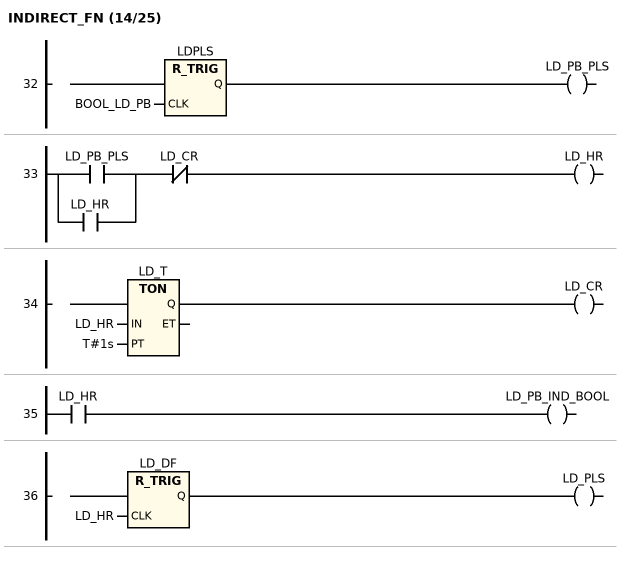
// NETWORK 32
LDPLS(CLK := BOOL_LD_PB); // R_TRIG
LD_PB_PLS := LDPLS.Q;

// NETWORK 33
LD_HR := (LD_PB_PLS OR LD_HR) AND NOT LD_CR;

// NETWORK 34
LD_T(IN := LD_HR, PT := T#1s); // TON
LD_CR := LD_T.Q;

// NETWORK 35
LD_PB_IND_BOOL := LD_HR;

// NETWORK 36
LD_DF(CLK := LD_HR); // R_TRIG
LD_PLS := LD_DF.Q;

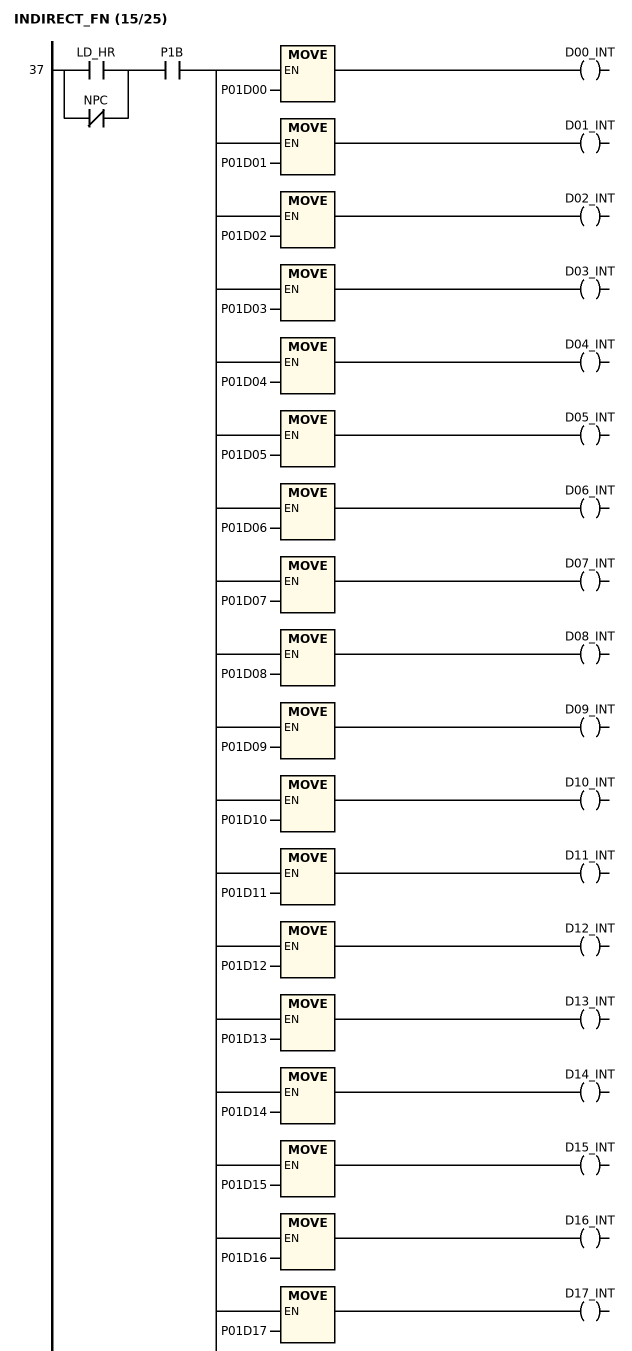
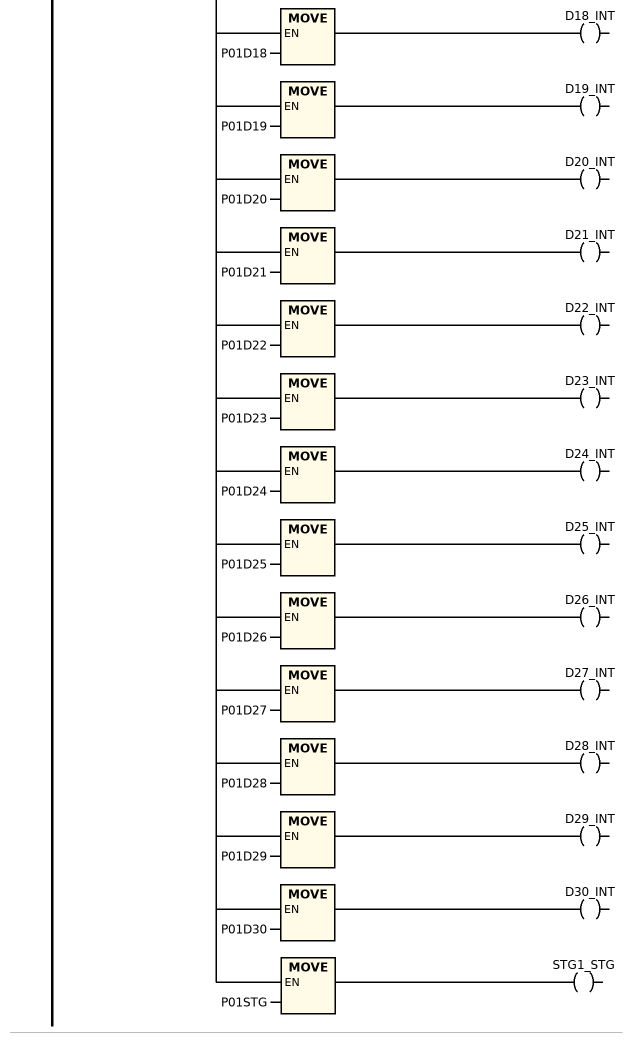
// NETWORK 37
_w365 := (LD_HR OR NOT NPC) AND P1B;
IF _w365 THEN _w366 := P01D00; END_IF
D00_INT := _w366;
IF _w365 THEN _w367 := P01D01; END_IF
D01_INT := _w367;
IF _w365 THEN _w368 := P01D02; END_IF
D02_INT := _w368;
IF _w365 THEN _w369 := P01D03; END_IF
D03_INT := _w369;
IF _w365 THEN _w370 := P01D04; END_IF
D04_INT := _w370;
IF _w365 THEN _w371 := P01D05; END_IF
D05_INT := _w371;
IF _w365 THEN _w372 := P01D06; END_IF
D06_INT := _w372;
IF _w365 THEN _w373 := P01D07; END_IF
D07_INT := _w373;
IF _w365 THEN _w374 := P01D08; END_IF
D08_INT := _w374;
IF _w365 THEN _w375 := P01D09; END_IF
D09_INT := _w375;
IF _w365 THEN _w376 := P01D10; END_IF
D10_INT := _w376;
IF _w365 THEN _w377 := P01D11; END_IF
D11_INT := _w377;
IF _w365 THEN _w378 := P01D12; END_IF
D12_INT := _w378;
IF _w365 THEN _w379 := P01D13; END_IF
D13_INT := _w379;
IF _w365 THEN _w380 := P01D14; END_IF
D14_INT := _w380;
IF _w365 THEN _w381 := P01D15; END_IF
D15_INT := _w381;
IF _w365 THEN _w382 := P01D16; END_IF
D16_INT := _w382;
IF _w365 THEN _w383 := P01D17; END_IF
D17_INT := _w383;
IF _w365 THEN _w384 := P01D18; END_IF
D18_INT := _w384;
IF _w365 THEN _w385 := P01D19; END_IF
D19_INT := _w385;
IF _w365 THEN _w386 := P01D20; END_IF
D20_INT := _w386;
IF _w365 THEN _w387 := P01D21; END_IF
D21_INT := _w387;
IF _w365 THEN _w388 := P01D22; END_IF
D22_INT := _w388;
IF _w365 THEN _w389 := P01D23; END_IF
D23_INT := _w389;
IF _w365 THEN _w390 := P01D24; END_IF
D24_INT := _w390;
IF _w365 THEN _w391 := P01D25; END_IF
D25_INT := _w391;
IF _w365 THEN _w392 := P01D26; END_IF
D26_INT := _w392;
IF _w365 THEN _w393 := P01D27; END_IF
D27_INT := _w393;
IF _w365 THEN _w394 := P01D28; END_IF
D28_INT := _w394;
IF _w365 THEN _w395 := P01D29; END_IF
D29_INT := _w395;
IF _w365 THEN _w396 := P01D30; END_IF
D30_INT := _w396;
IF _w365 THEN _w397 := P01STG; END_IF
STG1_STG := _w397;

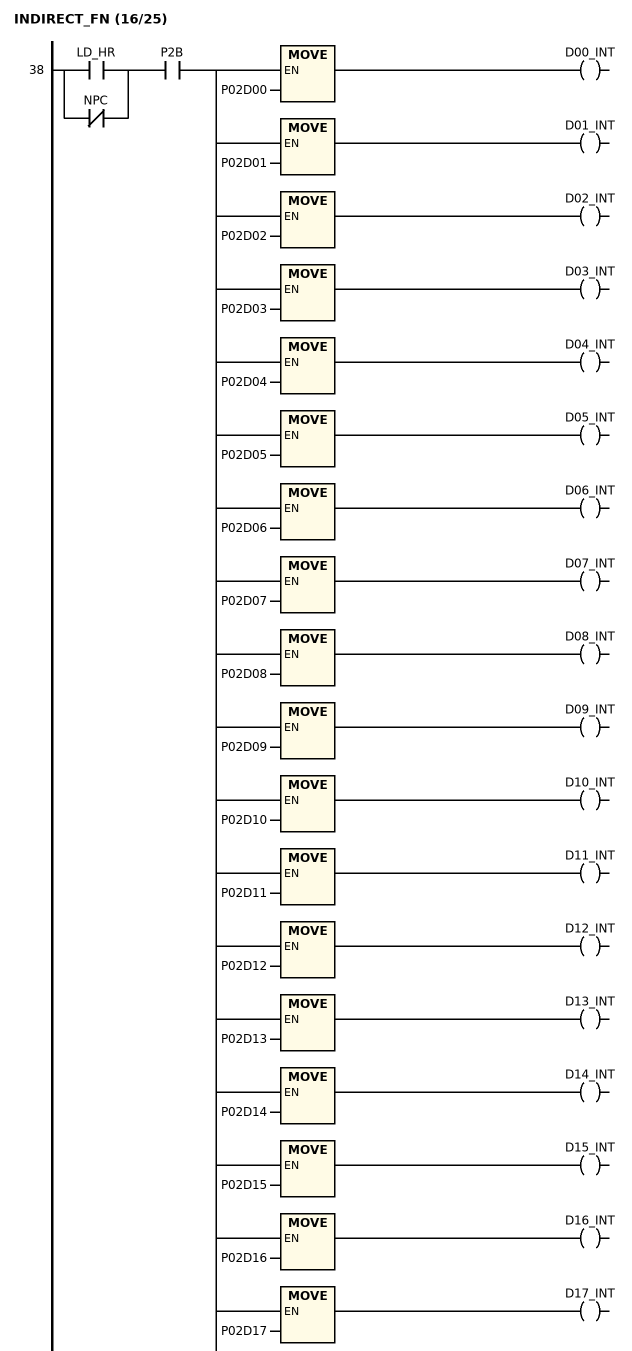
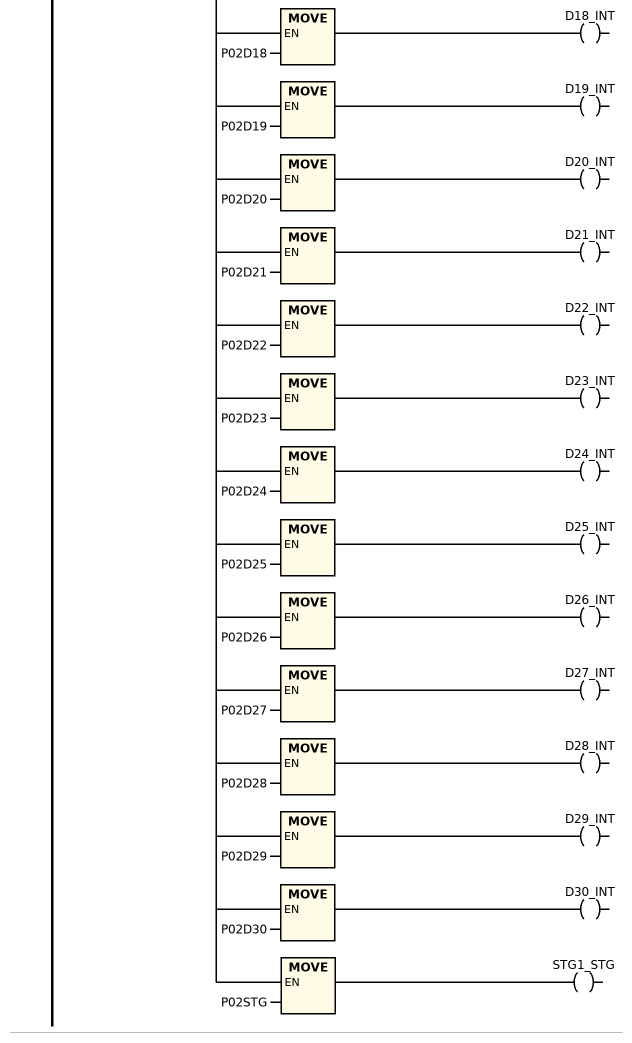
// NETWORK 38
_w398 := (LD_HR OR NOT NPC) AND P2B;
IF _w398 THEN _w399 := P02D00; END_IF
D00_INT := _w399;
IF _w398 THEN _w400 := P02D01; END_IF
D01_INT := _w400;
IF _w398 THEN _w401 := P02D02; END_IF
D02_INT := _w401;
IF _w398 THEN _w402 := P02D03; END_IF
D03_INT := _w402;
IF _w398 THEN _w403 := P02D04; END_IF
D04_INT := _w403;
IF _w398 THEN _w404 := P02D05; END_IF
D05_INT := _w404;
IF _w398 THEN _w405 := P02D06; END_IF
D06_INT := _w405;
IF _w398 THEN _w406 := P02D07; END_IF
D07_INT := _w406;
IF _w398 THEN _w407 := P02D08; END_IF
D08_INT := _w407;
IF _w398 THEN _w408 := P02D09; END_IF
D09_INT := _w408;
IF _w398 THEN _w409 := P02D10; END_IF
D10_INT := _w409;
IF _w398 THEN _w410 := P02D11; END_IF
D11_INT := _w410;
IF _w398 THEN _w411 := P02D12; END_IF
D12_INT := _w411;
IF _w398 THEN _w412 := P02D13; END_IF
D13_INT := _w412;
IF _w398 THEN _w413 := P02D14; END_IF
D14_INT := _w413;
IF _w398 THEN _w414 := P02D15; END_IF
D15_INT := _w414;
IF _w398 THEN _w415 := P02D16; END_IF
D16_INT := _w415;
IF _w398 THEN _w416 := P02D17; END_IF
D17_INT := _w416;
IF _w398 THEN _w417 := P02D18; END_IF
D18_INT := _w417;
IF _w398 THEN _w418 := P02D19; END_IF
D19_INT := _w418;
IF _w398 THEN _w419 := P02D20; END_IF
D20_INT := _w419;
IF _w398 THEN _w420 := P02D21; END_IF
D21_INT := _w420;
IF _w398 THEN _w421 := P02D22; END_IF
D22_INT := _w421;
IF _w398 THEN _w422 := P02D23; END_IF
D23_INT := _w422;
IF _w398 THEN _w423 := P02D24; END_IF
D24_INT := _w423;
IF _w398 THEN _w424 := P02D25; END_IF
D25_INT := _w424;
IF _w398 THEN _w425 := P02D26; END_IF
D26_INT := _w425;
IF _w398 THEN _w426 := P02D27; END_IF
D27_INT := _w426;
IF _w398 THEN _w427 := P02D28; END_IF
D28_INT := _w427;
IF _w398 THEN _w428 := P02D29; END_IF
D29_INT := _w428;
IF _w398 THEN _w429 := P02D30; END_IF
D30_INT := _w429;
IF _w398 THEN _w430 := P02STG; END_IF
STG1_STG := _w430;

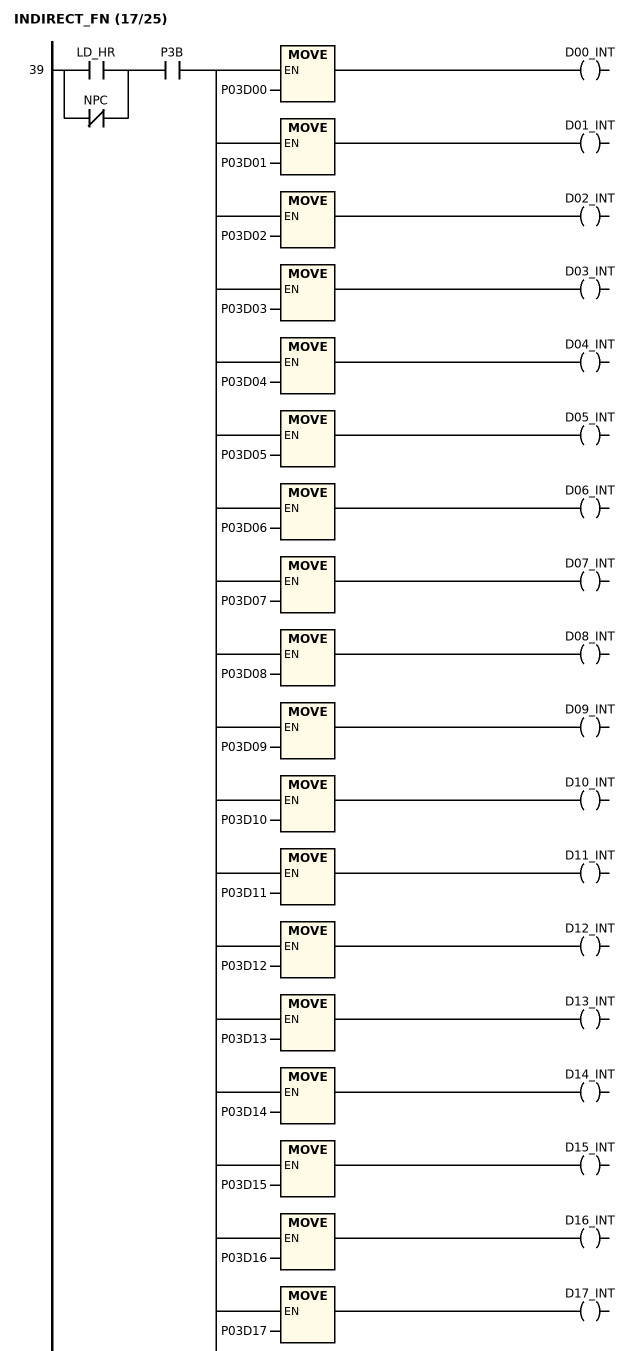
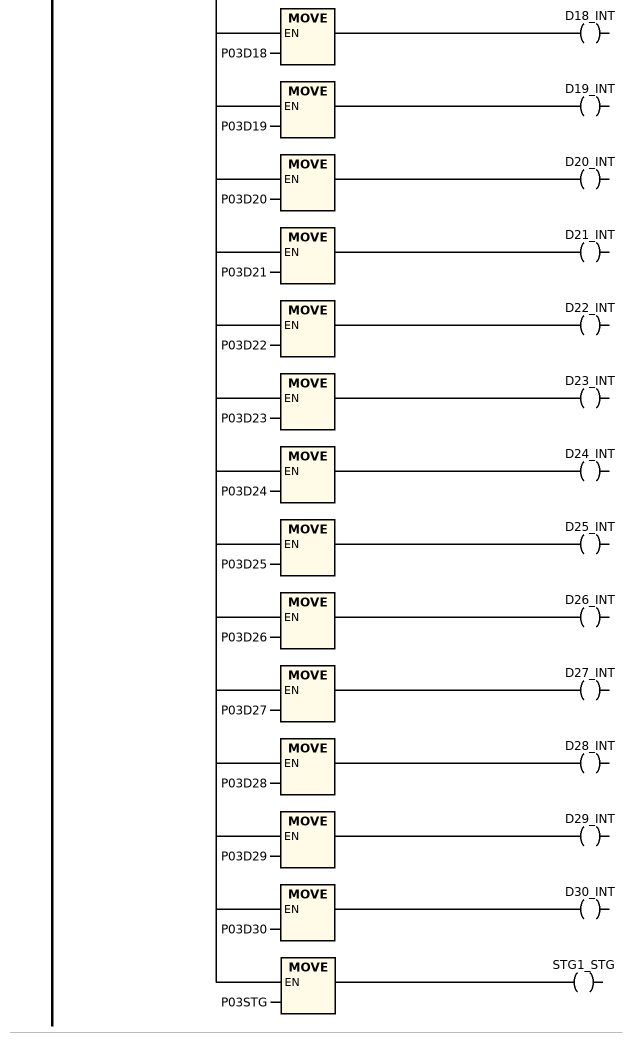
// NETWORK 39
_w431 := (LD_HR OR NOT NPC) AND P3B;
IF _w431 THEN _w432 := P03D00; END_IF
D00_INT := _w432;
IF _w431 THEN _w433 := P03D01; END_IF
D01_INT := _w433;
IF _w431 THEN _w434 := P03D02; END_IF
D02_INT := _w434;
IF _w431 THEN _w435 := P03D03; END_IF
D03_INT := _w435;
IF _w431 THEN _w436 := P03D04; END_IF
D04_INT := _w436;
IF _w431 THEN _w437 := P03D05; END_IF
D05_INT := _w437;
IF _w431 THEN _w438 := P03D06; END_IF
D06_INT := _w438;
IF _w431 THEN _w439 := P03D07; END_IF
D07_INT := _w439;
IF _w431 THEN _w440 := P03D08; END_IF
D08_INT := _w440;
IF _w431 THEN _w441 := P03D09; END_IF
D09_INT := _w441;
IF _w431 THEN _w442 := P03D10; END_IF
D10_INT := _w442;
IF _w431 THEN _w443 := P03D11; END_IF
D11_INT := _w443;
IF _w431 THEN _w444 := P03D12; END_IF
D12_INT := _w444;
IF _w431 THEN _w445 := P03D13; END_IF
D13_INT := _w445;
IF _w431 THEN _w446 := P03D14; END_IF
D14_INT := _w446;
IF _w431 THEN _w447 := P03D15; END_IF
D15_INT := _w447;
IF _w431 THEN _w448 := P03D16; END_IF
D16_INT := _w448;
IF _w431 THEN _w449 := P03D17; END_IF
D17_INT := _w449;
IF _w431 THEN _w450 := P03D18; END_IF
D18_INT := _w450;
IF _w431 THEN _w451 := P03D19; END_IF
D19_INT := _w451;
IF _w431 THEN _w452 := P03D20; END_IF
D20_INT := _w452;
IF _w431 THEN _w453 := P03D21; END_IF
D21_INT := _w453;
IF _w431 THEN _w454 := P03D22; END_IF
D22_INT := _w454;
IF _w431 THEN _w455 := P03D23; END_IF
D23_INT := _w455;
IF _w431 THEN _w456 := P03D24; END_IF
D24_INT := _w456;
IF _w431 THEN _w457 := P03D25; END_IF
D25_INT := _w457;
IF _w431 THEN _w458 := P03D26; END_IF
D26_INT := _w458;
IF _w431 THEN _w459 := P03D27; END_IF
D27_INT := _w459;
IF _w431 THEN _w460 := P03D28; END_IF
D28_INT := _w460;
IF _w431 THEN _w461 := P03D29; END_IF
D29_INT := _w461;
IF _w431 THEN _w462 := P03D30; END_IF
D30_INT := _w462;
IF _w431 THEN _w463 := P03STG; END_IF
STG1_STG := _w463;

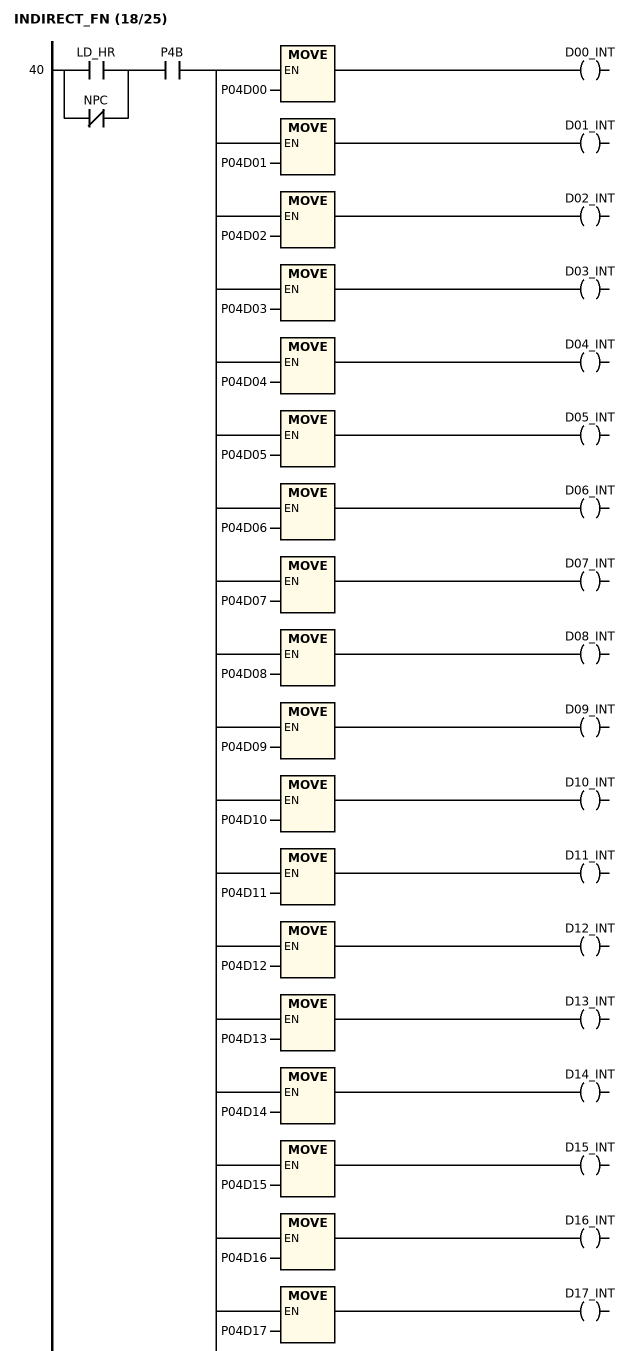
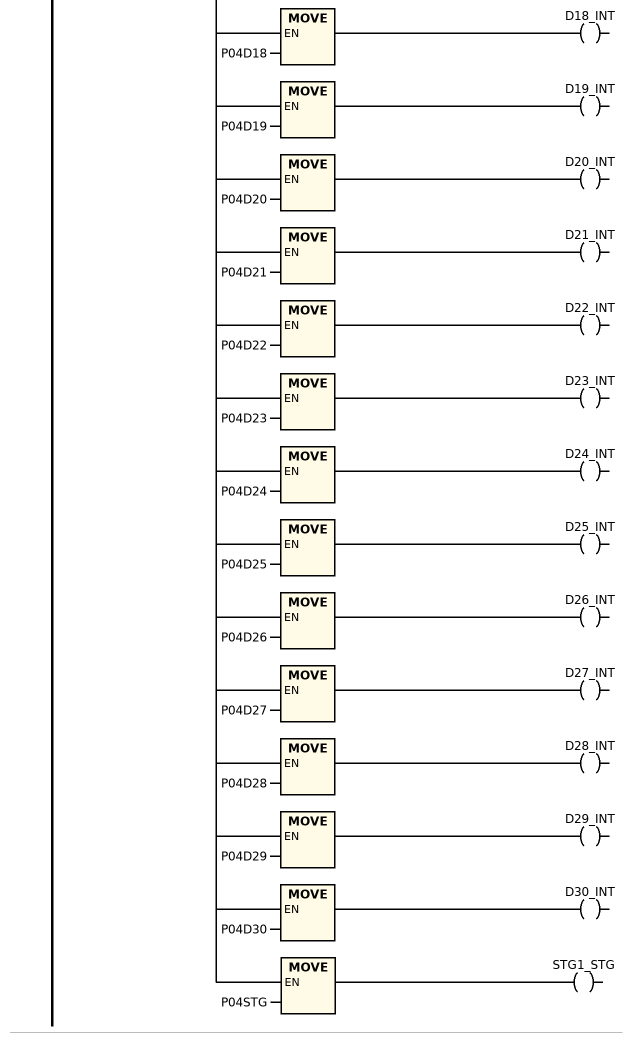
// NETWORK 40
_w464 := (LD_HR OR NOT NPC) AND P4B;
IF _w464 THEN _w465 := P04D00; END_IF
D00_INT := _w465;
IF _w464 THEN _w466 := P04D01; END_IF
D01_INT := _w466;
IF _w464 THEN _w467 := P04D02; END_IF
D02_INT := _w467;
IF _w464 THEN _w468 := P04D03; END_IF
D03_INT := _w468;
IF _w464 THEN _w469 := P04D04; END_IF
D04_INT := _w469;
IF _w464 THEN _w470 := P04D05; END_IF
D05_INT := _w470;
IF _w464 THEN _w471 := P04D06; END_IF
D06_INT := _w471;
IF _w464 THEN _w472 := P04D07; END_IF
D07_INT := _w472;
IF _w464 THEN _w473 := P04D08; END_IF
D08_INT := _w473;
IF _w464 THEN _w474 := P04D09; END_IF
D09_INT := _w474;
IF _w464 THEN _w475 := P04D10; END_IF
D10_INT := _w475;
IF _w464 THEN _w476 := P04D11; END_IF
D11_INT := _w476;
IF _w464 THEN _w477 := P04D12; END_IF
D12_INT := _w477;
IF _w464 THEN _w478 := P04D13; END_IF
D13_INT := _w478;
IF _w464 THEN _w479 := P04D14; END_IF
D14_INT := _w479;
IF _w464 THEN _w480 := P04D15; END_IF
D15_INT := _w480;
IF _w464 THEN _w481 := P04D16; END_IF
D16_INT := _w481;
IF _w464 THEN _w482 := P04D17; END_IF
D17_INT := _w482;
IF _w464 THEN _w483 := P04D18; END_IF
D18_INT := _w483;
IF _w464 THEN _w484 := P04D19; END_IF
D19_INT := _w484;
IF _w464 THEN _w485 := P04D20; END_IF
D20_INT := _w485;
IF _w464 THEN _w486 := P04D21; END_IF
D21_INT := _w486;
IF _w464 THEN _w487 := P04D22; END_IF
D22_INT := _w487;
IF _w464 THEN _w488 := P04D23; END_IF
D23_INT := _w488;
IF _w464 THEN _w489 := P04D24; END_IF
D24_INT := _w489;
IF _w464 THEN _w490 := P04D25; END_IF
D25_INT := _w490;
IF _w464 THEN _w491 := P04D26; END_IF
D26_INT := _w491;
IF _w464 THEN _w492 := P04D27; END_IF
D27_INT := _w492;
IF _w464 THEN _w493 := P04D28; END_IF
D28_INT := _w493;
IF _w464 THEN _w494 := P04D29; END_IF
D29_INT := _w494;
IF _w464 THEN _w495 := P04D30; END_IF
D30_INT := _w495;
IF _w464 THEN _w496 := P04STG; END_IF
STG1_STG := _w496;

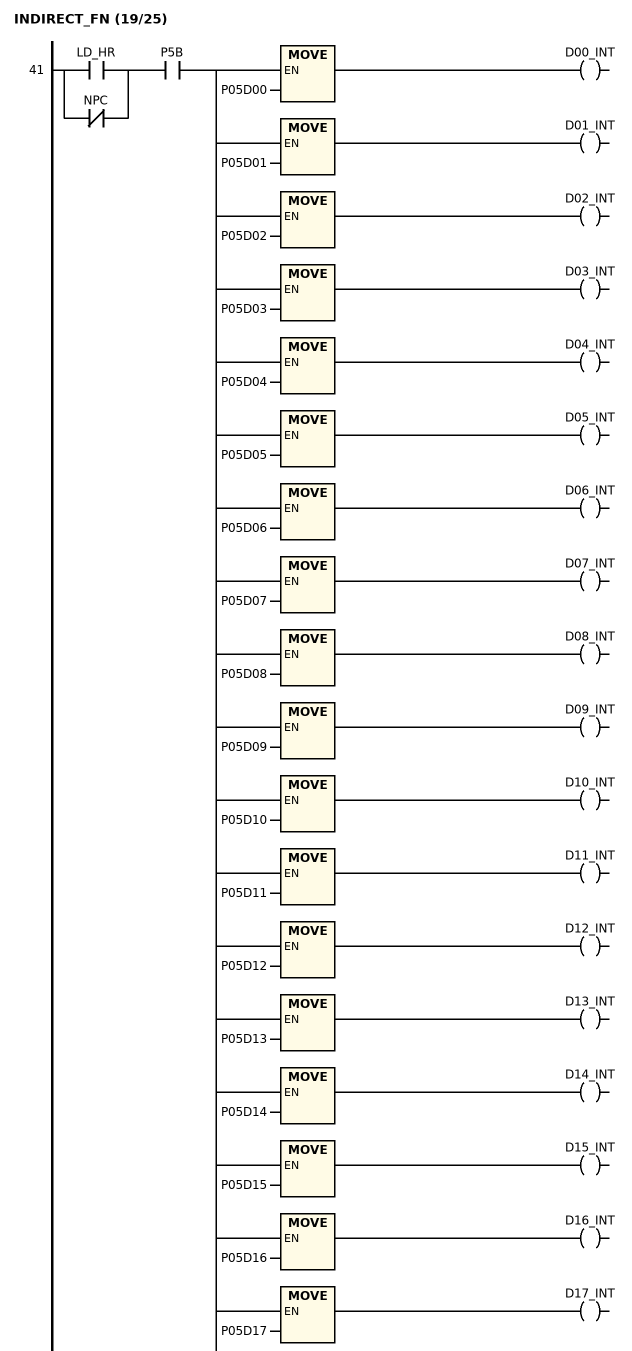
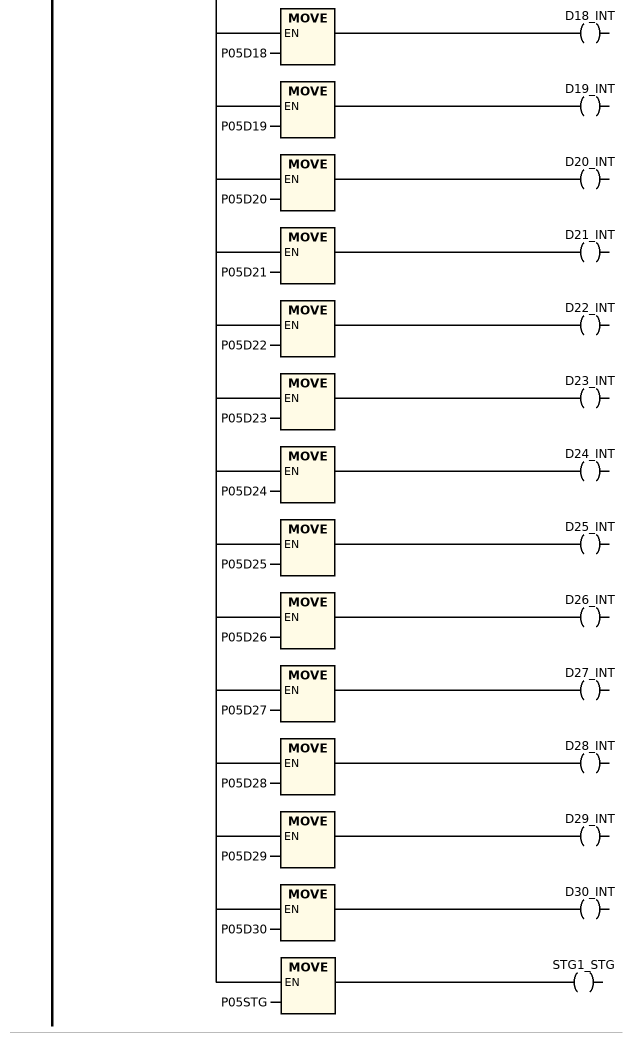
// NETWORK 41
_w497 := (LD_HR OR NOT NPC) AND P5B;
IF _w497 THEN _w498 := P05D00; END_IF
D00_INT := _w498;
IF _w497 THEN _w499 := P05D01; END_IF
D01_INT := _w499;
IF _w497 THEN _w500 := P05D02; END_IF
D02_INT := _w500;
IF _w497 THEN _w501 := P05D03; END_IF
D03_INT := _w501;
IF _w497 THEN _w502 := P05D04; END_IF
D04_INT := _w502;
IF _w497 THEN _w503 := P05D05; END_IF
D05_INT := _w503;
IF _w497 THEN _w504 := P05D06; END_IF
D06_INT := _w504;
IF _w497 THEN _w505 := P05D07; END_IF
D07_INT := _w505;
IF _w497 THEN _w506 := P05D08; END_IF
D08_INT := _w506;
IF _w497 THEN _w507 := P05D09; END_IF
D09_INT := _w507;
IF _w497 THEN _w508 := P05D10; END_IF
D10_INT := _w508;
IF _w497 THEN _w509 := P05D11; END_IF
D11_INT := _w509;
IF _w497 THEN _w510 := P05D12; END_IF
D12_INT := _w510;
IF _w497 THEN _w511 := P05D13; END_IF
D13_INT := _w511;
IF _w497 THEN _w512 := P05D14; END_IF
D14_INT := _w512;
IF _w497 THEN _w513 := P05D15; END_IF
D15_INT := _w513;
IF _w497 THEN _w514 := P05D16; END_IF
D16_INT := _w514;
IF _w497 THEN _w515 := P05D17; END_IF
D17_INT := _w515;
IF _w497 THEN _w516 := P05D18; END_IF
D18_INT := _w516;
IF _w497 THEN _w517 := P05D19; END_IF
D19_INT := _w517;
IF _w497 THEN _w518 := P05D20; END_IF
D20_INT := _w518;
IF _w497 THEN _w519 := P05D21; END_IF
D21_INT := _w519;
IF _w497 THEN _w520 := P05D22; END_IF
D22_INT := _w520;
IF _w497 THEN _w521 := P05D23; END_IF
D23_INT := _w521;
IF _w497 THEN _w522 := P05D24; END_IF
D24_INT := _w522;
IF _w497 THEN _w523 := P05D25; END_IF
D25_INT := _w523;
IF _w497 THEN _w524 := P05D26; END_IF
D26_INT := _w524;
IF _w497 THEN _w525 := P05D27; END_IF
D27_INT := _w525;
IF _w497 THEN _w526 := P05D28; END_IF
D28_INT := _w526;
IF _w497 THEN _w527 := P05D29; END_IF
D29_INT := _w527;
IF _w497 THEN _w528 := P05D30; END_IF
D30_INT := _w528;
IF _w497 THEN _w529 := P05STG; END_IF
STG1_STG := _w529;

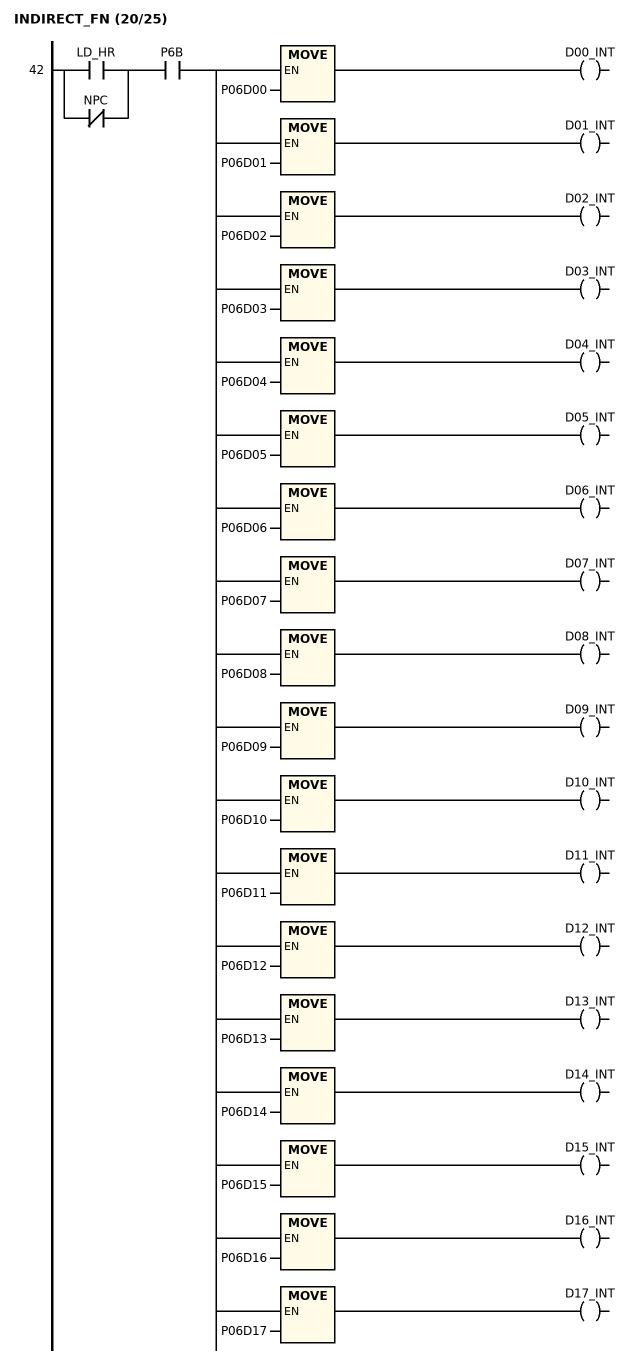
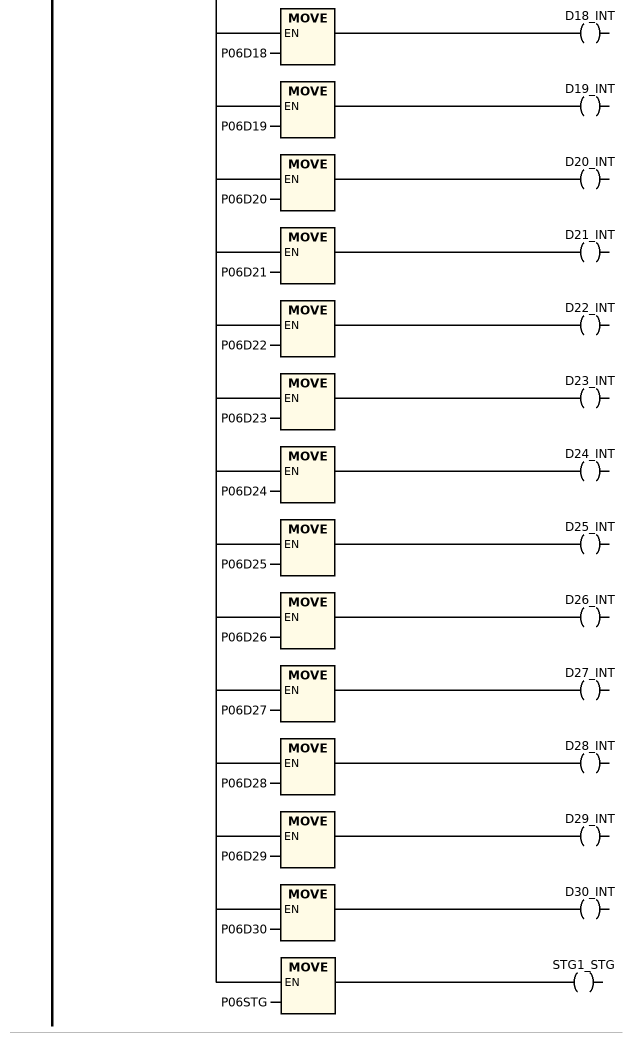
// NETWORK 42
_w530 := (LD_HR OR NOT NPC) AND P6B;
IF _w530 THEN _w531 := P06D00; END_IF
D00_INT := _w531;
IF _w530 THEN _w532 := P06D01; END_IF
D01_INT := _w532;
IF _w530 THEN _w533 := P06D02; END_IF
D02_INT := _w533;
IF _w530 THEN _w534 := P06D03; END_IF
D03_INT := _w534;
IF _w530 THEN _w535 := P06D04; END_IF
D04_INT := _w535;
IF _w530 THEN _w536 := P06D05; END_IF
D05_INT := _w536;
IF _w530 THEN _w537 := P06D06; END_IF
D06_INT := _w537;
IF _w530 THEN _w538 := P06D07; END_IF
D07_INT := _w538;
IF _w530 THEN _w539 := P06D08; END_IF
D08_INT := _w539;
IF _w530 THEN _w540 := P06D09; END_IF
D09_INT := _w540;
IF _w530 THEN _w541 := P06D10; END_IF
D10_INT := _w541;
IF _w530 THEN _w542 := P06D11; END_IF
D11_INT := _w542;
IF _w530 THEN _w543 := P06D12; END_IF
D12_INT := _w543;
IF _w530 THEN _w544 := P06D13; END_IF
D13_INT := _w544;
IF _w530 THEN _w545 := P06D14; END_IF
D14_INT := _w545;
IF _w530 THEN _w546 := P06D15; END_IF
D15_INT := _w546;
IF _w530 THEN _w547 := P06D16; END_IF
D16_INT := _w547;
IF _w530 THEN _w548 := P06D17; END_IF
D17_INT := _w548;
IF _w530 THEN _w549 := P06D18; END_IF
D18_INT := _w549;
IF _w530 THEN _w550 := P06D19; END_IF
D19_INT := _w550;
IF _w530 THEN _w551 := P06D20; END_IF
D20_INT := _w551;
IF _w530 THEN _w552 := P06D21; END_IF
D21_INT := _w552;
IF _w530 THEN _w553 := P06D22; END_IF
D22_INT := _w553;
IF _w530 THEN _w554 := P06D23; END_IF
D23_INT := _w554;
IF _w530 THEN _w555 := P06D24; END_IF
D24_INT := _w555;
IF _w530 THEN _w556 := P06D25; END_IF
D25_INT := _w556;
IF _w530 THEN _w557 := P06D26; END_IF
D26_INT := _w557;
IF _w530 THEN _w558 := P06D27; END_IF
D27_INT := _w558;
IF _w530 THEN _w559 := P06D28; END_IF
D28_INT := _w559;
IF _w530 THEN _w560 := P06D29; END_IF
D29_INT := _w560;
IF _w530 THEN _w561 := P06D30; END_IF
D30_INT := _w561;
IF _w530 THEN _w562 := P06STG; END_IF
STG1_STG := _w562;

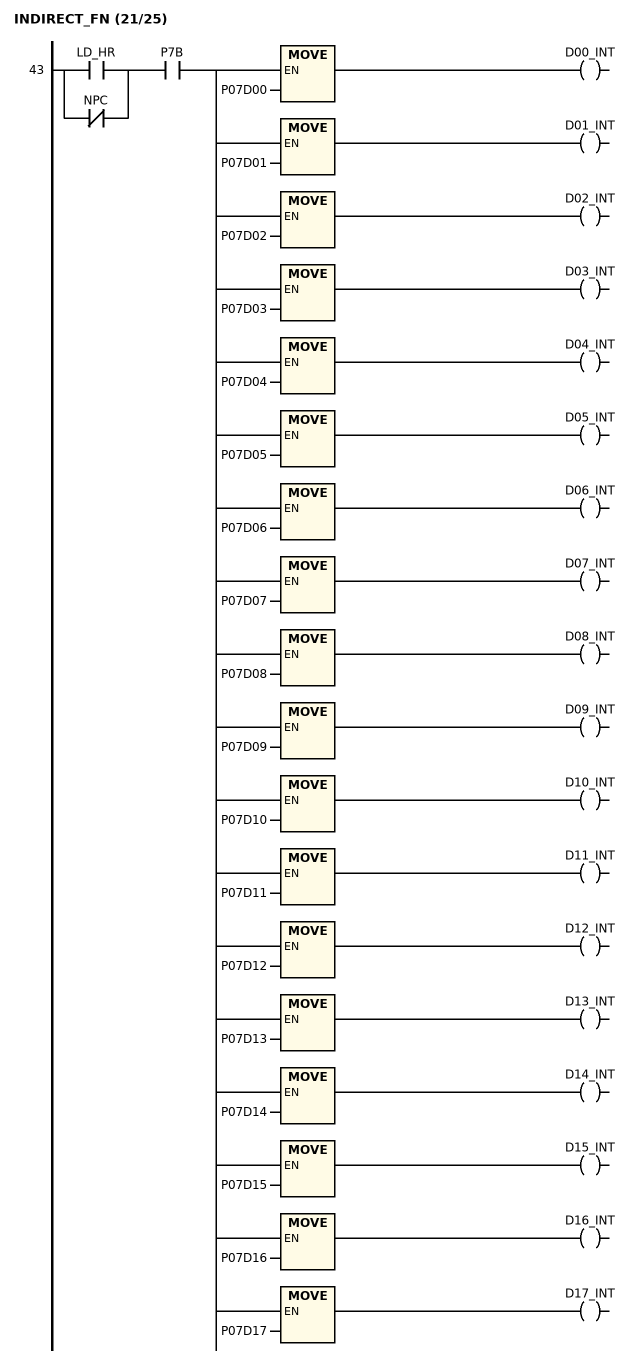
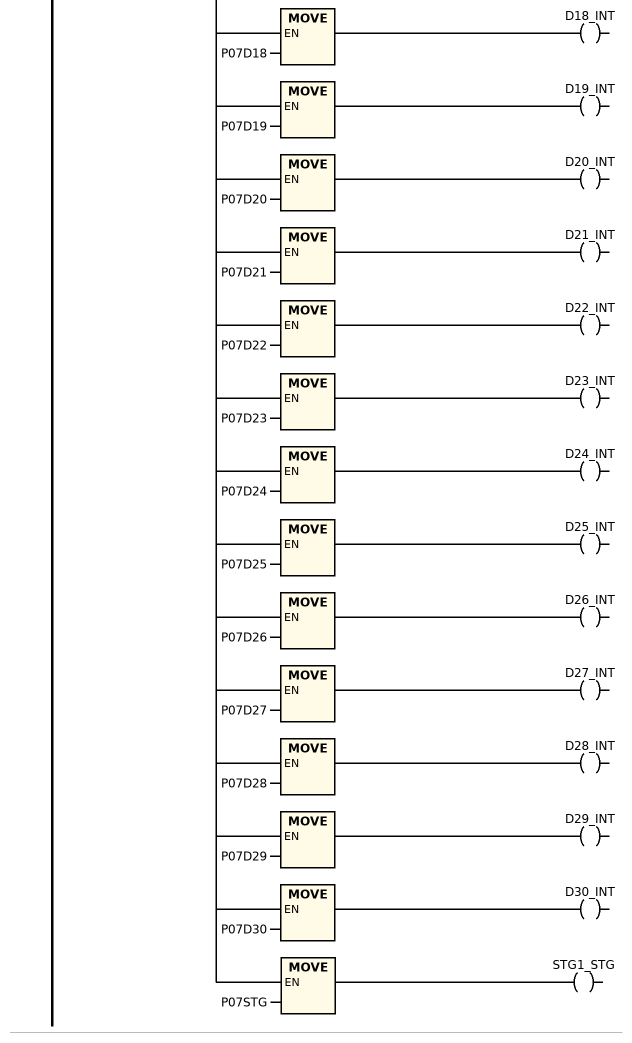
// NETWORK 43
_w563 := (LD_HR OR NOT NPC) AND P7B;
IF _w563 THEN _w564 := P07D00; END_IF
D00_INT := _w564;
IF _w563 THEN _w565 := P07D01; END_IF
D01_INT := _w565;
IF _w563 THEN _w566 := P07D02; END_IF
D02_INT := _w566;
IF _w563 THEN _w567 := P07D03; END_IF
D03_INT := _w567;
IF _w563 THEN _w568 := P07D04; END_IF
D04_INT := _w568;
IF _w563 THEN _w569 := P07D05; END_IF
D05_INT := _w569;
IF _w563 THEN _w570 := P07D06; END_IF
D06_INT := _w570;
IF _w563 THEN _w571 := P07D07; END_IF
D07_INT := _w571;
IF _w563 THEN _w572 := P07D08; END_IF
D08_INT := _w572;
IF _w563 THEN _w573 := P07D09; END_IF
D09_INT := _w573;
IF _w563 THEN _w574 := P07D10; END_IF
D10_INT := _w574;
IF _w563 THEN _w575 := P07D11; END_IF
D11_INT := _w575;
IF _w563 THEN _w576 := P07D12; END_IF
D12_INT := _w576;
IF _w563 THEN _w577 := P07D13; END_IF
D13_INT := _w577;
IF _w563 THEN _w578 := P07D14; END_IF
D14_INT := _w578;
IF _w563 THEN _w579 := P07D15; END_IF
D15_INT := _w579;
IF _w563 THEN _w580 := P07D16; END_IF
D16_INT := _w580;
IF _w563 THEN _w581 := P07D17; END_IF
D17_INT := _w581;
IF _w563 THEN _w582 := P07D18; END_IF
D18_INT := _w582;
IF _w563 THEN _w583 := P07D19; END_IF
D19_INT := _w583;
IF _w563 THEN _w584 := P07D20; END_IF
D20_INT := _w584;
IF _w563 THEN _w585 := P07D21; END_IF
D21_INT := _w585;
IF _w563 THEN _w586 := P07D22; END_IF
D22_INT := _w586;
IF _w563 THEN _w587 := P07D23; END_IF
D23_INT := _w587;
IF _w563 THEN _w588 := P07D24; END_IF
D24_INT := _w588;
IF _w563 THEN _w589 := P07D25; END_IF
D25_INT := _w589;
IF _w563 THEN _w590 := P07D26; END_IF
D26_INT := _w590;
IF _w563 THEN _w591 := P07D27; END_IF
D27_INT := _w591;
IF _w563 THEN _w592 := P07D28; END_IF
D28_INT := _w592;
IF _w563 THEN _w593 := P07D29; END_IF
D29_INT := _w593;
IF _w563 THEN _w594 := P07D30; END_IF
D30_INT := _w594;
IF _w563 THEN _w595 := P07STG; END_IF
STG1_STG := _w595;

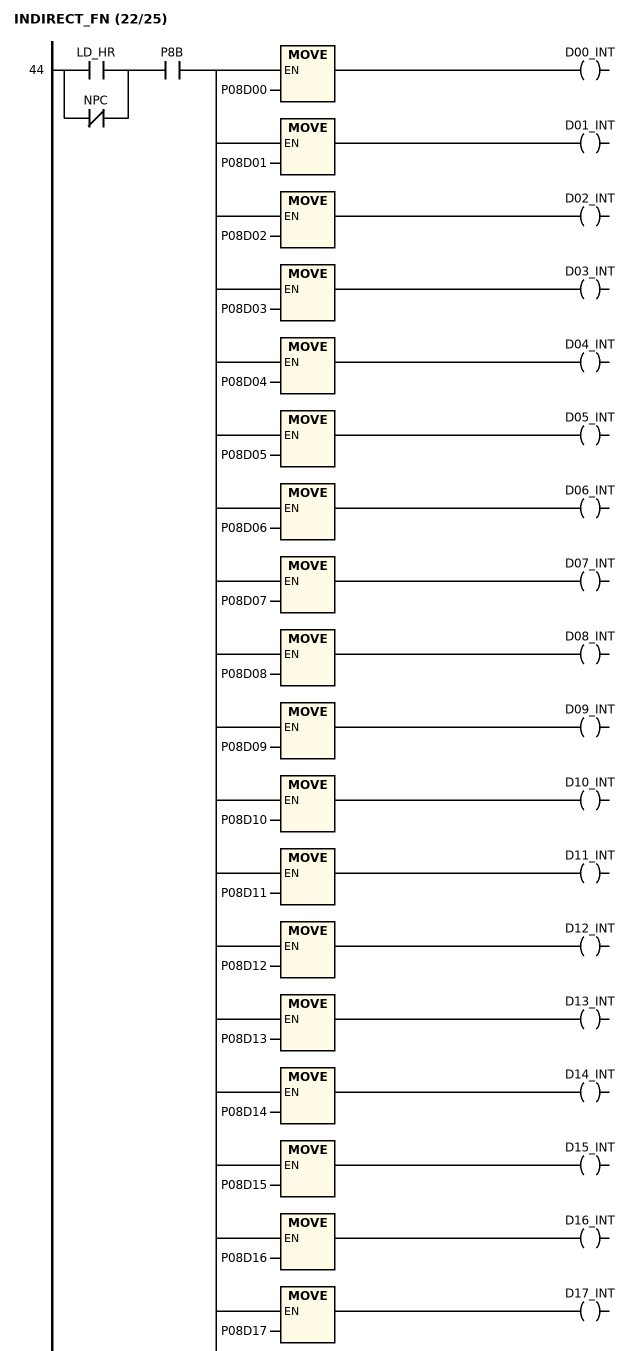
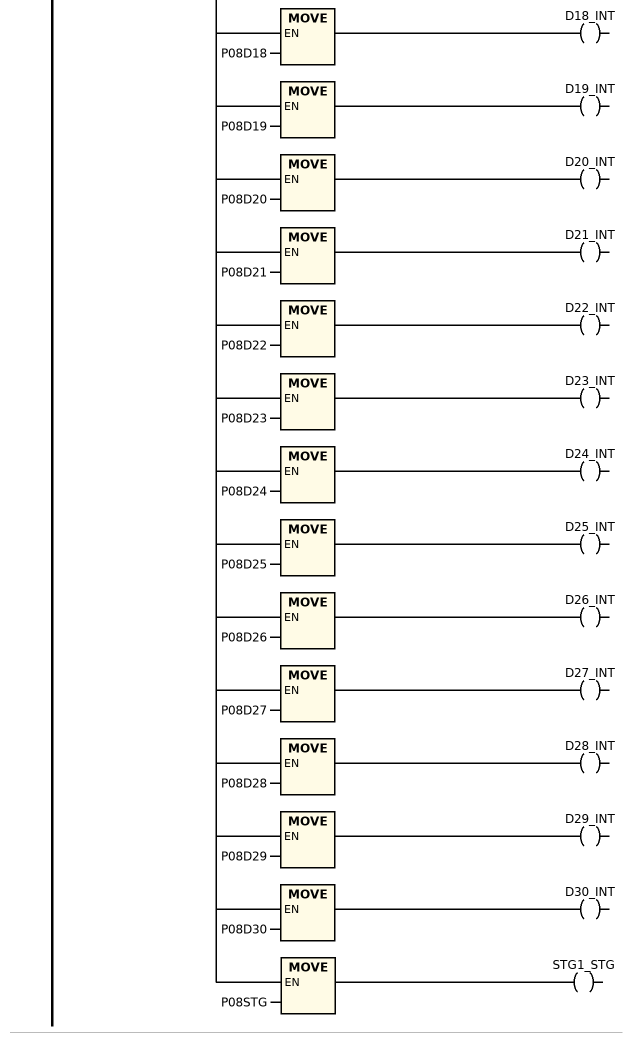
// NETWORK 44
_w596 := (LD_HR OR NOT NPC) AND P8B;
IF _w596 THEN _w597 := P08D00; END_IF
D00_INT := _w597;
IF _w596 THEN _w598 := P08D01; END_IF
D01_INT := _w598;
IF _w596 THEN _w599 := P08D02; END_IF
D02_INT := _w599;
IF _w596 THEN _w600 := P08D03; END_IF
D03_INT := _w600;
IF _w596 THEN _w601 := P08D04; END_IF
D04_INT := _w601;
IF _w596 THEN _w602 := P08D05; END_IF
D05_INT := _w602;
IF _w596 THEN _w603 := P08D06; END_IF
D06_INT := _w603;
IF _w596 THEN _w604 := P08D07; END_IF
D07_INT := _w604;
IF _w596 THEN _w605 := P08D08; END_IF
D08_INT := _w605;
IF _w596 THEN _w606 := P08D09; END_IF
D09_INT := _w606;
IF _w596 THEN _w607 := P08D10; END_IF
D10_INT := _w607;
IF _w596 THEN _w608 := P08D11; END_IF
D11_INT := _w608;
IF _w596 THEN _w609 := P08D12; END_IF
D12_INT := _w609;
IF _w596 THEN _w610 := P08D13; END_IF
D13_INT := _w610;
IF _w596 THEN _w611 := P08D14; END_IF
D14_INT := _w611;
IF _w596 THEN _w612 := P08D15; END_IF
D15_INT := _w612;
IF _w596 THEN _w613 := P08D16; END_IF
D16_INT := _w613;
IF _w596 THEN _w614 := P08D17; END_IF
D17_INT := _w614;
IF _w596 THEN _w615 := P08D18; END_IF
D18_INT := _w615;
IF _w596 THEN _w616 := P08D19; END_IF
D19_INT := _w616;
IF _w596 THEN _w617 := P08D20; END_IF
D20_INT := _w617;
IF _w596 THEN _w618 := P08D21; END_IF
D21_INT := _w618;
IF _w596 THEN _w619 := P08D22; END_IF
D22_INT := _w619;
IF _w596 THEN _w620 := P08D23; END_IF
D23_INT := _w620;
IF _w596 THEN _w621 := P08D24; END_IF
D24_INT := _w621;
IF _w596 THEN _w622 := P08D25; END_IF
D25_INT := _w622;
IF _w596 THEN _w623 := P08D26; END_IF
D26_INT := _w623;
IF _w596 THEN _w624 := P08D27; END_IF
D27_INT := _w624;
IF _w596 THEN _w625 := P08D28; END_IF
D28_INT := _w625;
IF _w596 THEN _w626 := P08D29; END_IF
D29_INT := _w626;
IF _w596 THEN _w627 := P08D30; END_IF
D30_INT := _w627;
IF _w596 THEN _w628 := P08STG; END_IF
STG1_STG := _w628;

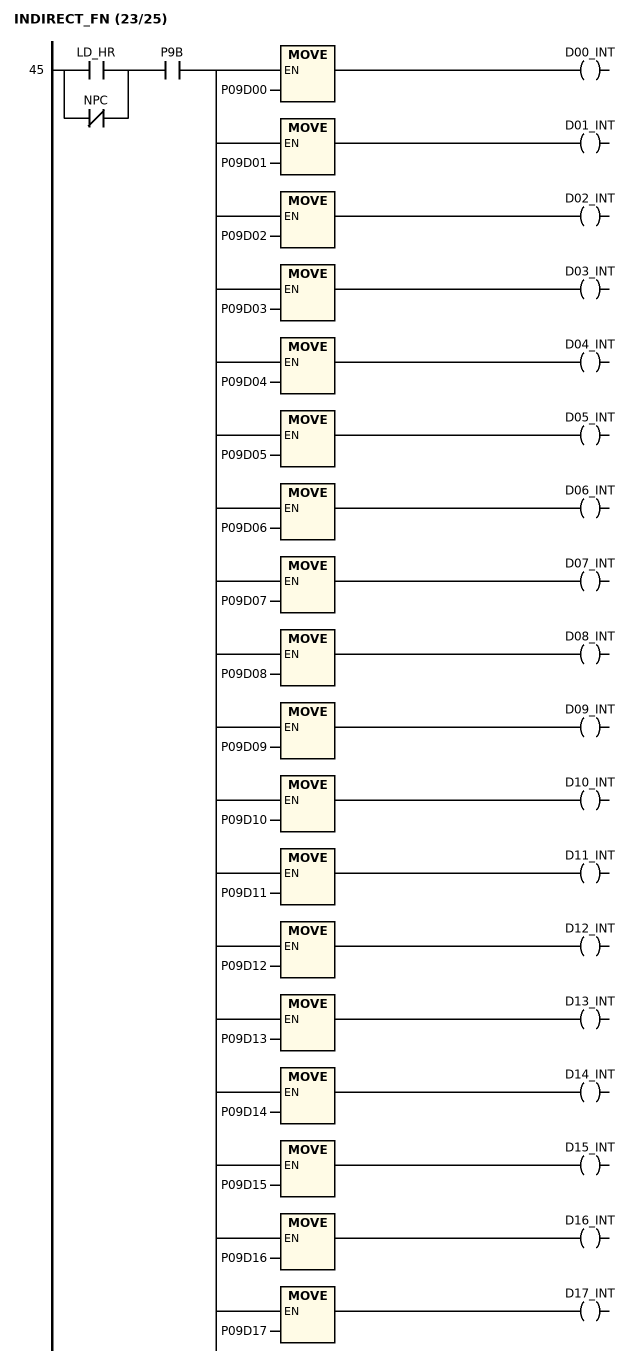
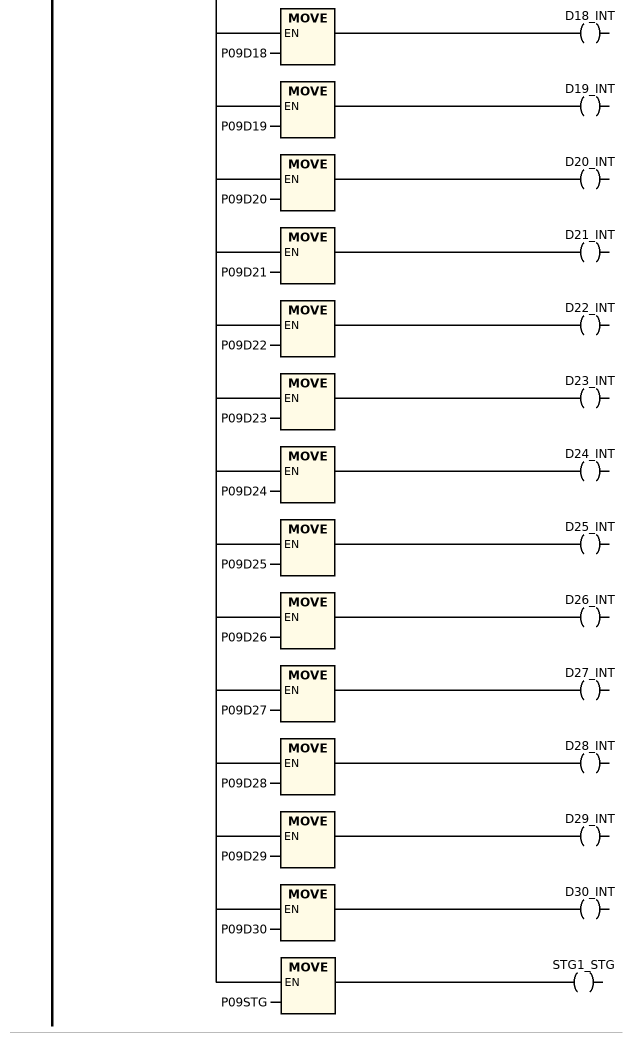
// NETWORK 45
_w629 := (LD_HR OR NOT NPC) AND P9B;
IF _w629 THEN _w630 := P09D00; END_IF
D00_INT := _w630;
IF _w629 THEN _w631 := P09D01; END_IF
D01_INT := _w631;
IF _w629 THEN _w632 := P09D02; END_IF
D02_INT := _w632;
IF _w629 THEN _w633 := P09D03; END_IF
D03_INT := _w633;
IF _w629 THEN _w634 := P09D04; END_IF
D04_INT := _w634;
IF _w629 THEN _w635 := P09D05; END_IF
D05_INT := _w635;
IF _w629 THEN _w636 := P09D06; END_IF
D06_INT := _w636;
IF _w629 THEN _w637 := P09D07; END_IF
D07_INT := _w637;
IF _w629 THEN _w638 := P09D08; END_IF
D08_INT := _w638;
IF _w629 THEN _w639 := P09D09; END_IF
D09_INT := _w639;
IF _w629 THEN _w640 := P09D10; END_IF
D10_INT := _w640;
IF _w629 THEN _w641 := P09D11; END_IF
D11_INT := _w641;
IF _w629 THEN _w642 := P09D12; END_IF
D12_INT := _w642;
IF _w629 THEN _w643 := P09D13; END_IF
D13_INT := _w643;
IF _w629 THEN _w644 := P09D14; END_IF
D14_INT := _w644;
IF _w629 THEN _w645 := P09D15; END_IF
D15_INT := _w645;
IF _w629 THEN _w646 := P09D16; END_IF
D16_INT := _w646;
IF _w629 THEN _w647 := P09D17; END_IF
D17_INT := _w647;
IF _w629 THEN _w648 := P09D18; END_IF
D18_INT := _w648;
IF _w629 THEN _w649 := P09D19; END_IF
D19_INT := _w649;
IF _w629 THEN _w650 := P09D20; END_IF
D20_INT := _w650;
IF _w629 THEN _w651 := P09D21; END_IF
D21_INT := _w651;
IF _w629 THEN _w652 := P09D22; END_IF
D22_INT := _w652;
IF _w629 THEN _w653 := P09D23; END_IF
D23_INT := _w653;
IF _w629 THEN _w654 := P09D24; END_IF
D24_INT := _w654;
IF _w629 THEN _w655 := P09D25; END_IF
D25_INT := _w655;
IF _w629 THEN _w656 := P09D26; END_IF
D26_INT := _w656;
IF _w629 THEN _w657 := P09D27; END_IF
D27_INT := _w657;
IF _w629 THEN _w658 := P09D28; END_IF
D28_INT := _w658;
IF _w629 THEN _w659 := P09D29; END_IF
D29_INT := _w659;
IF _w629 THEN _w660 := P09D30; END_IF
D30_INT := _w660;
IF _w629 THEN _w661 := P09STG; END_IF
STG1_STG := _w661;

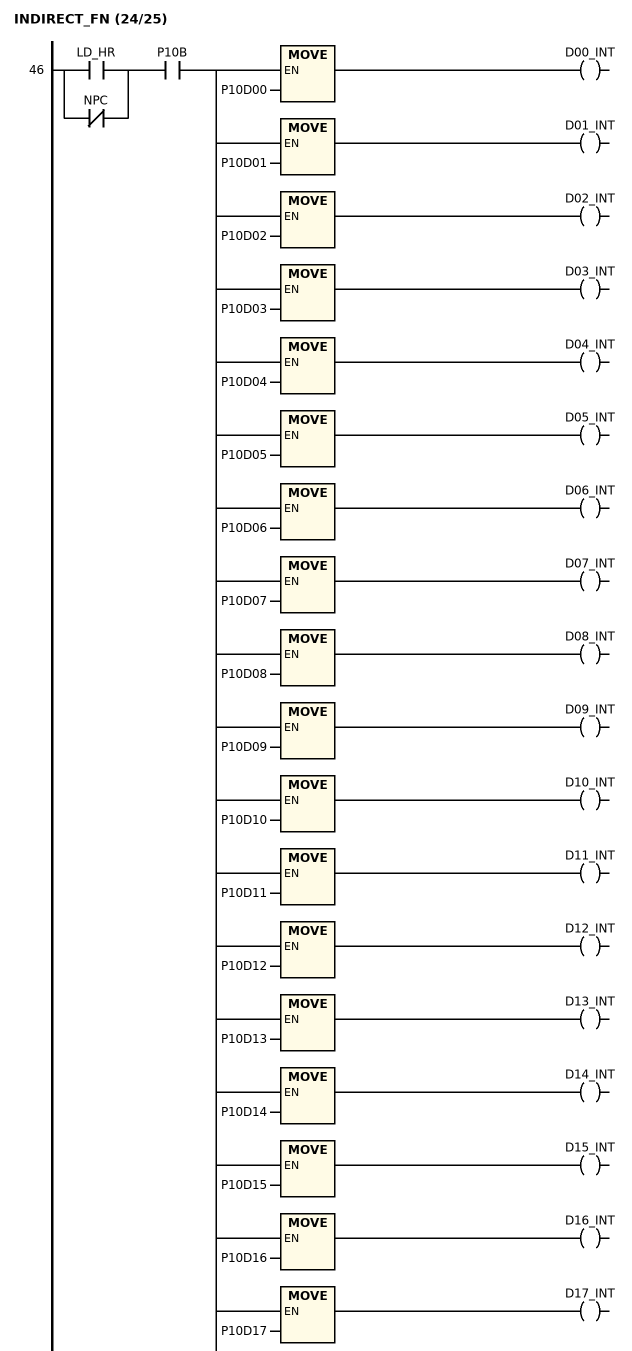
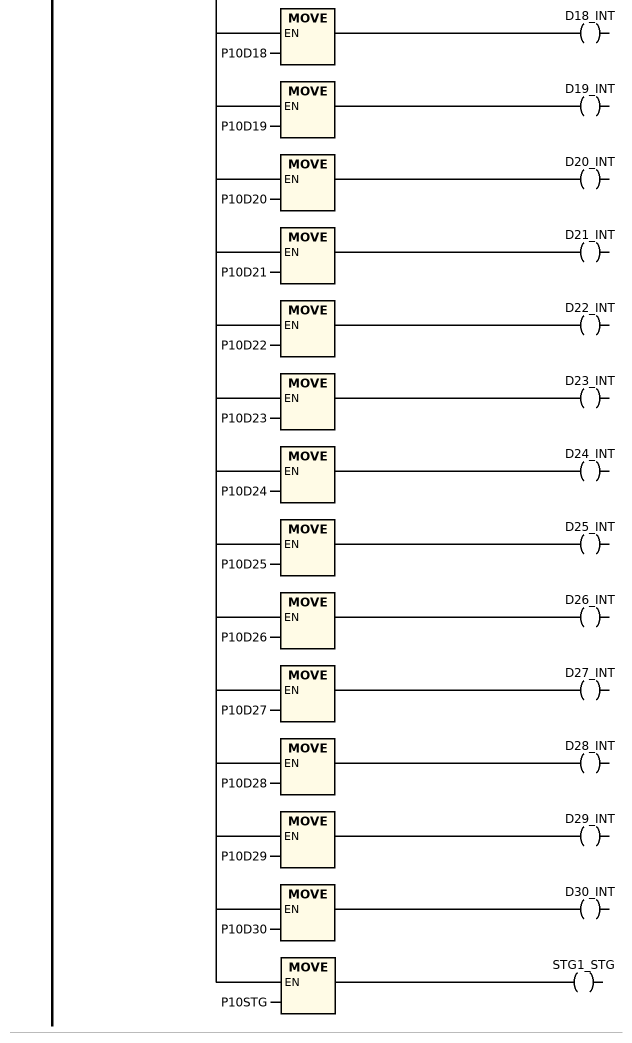
// NETWORK 46
_w662 := (LD_HR OR NOT NPC) AND P10B;
IF _w662 THEN _w663 := P10D00; END_IF
D00_INT := _w663;
IF _w662 THEN _w664 := P10D01; END_IF
D01_INT := _w664;
IF _w662 THEN _w665 := P10D02; END_IF
D02_INT := _w665;
IF _w662 THEN _w666 := P10D03; END_IF
D03_INT := _w666;
IF _w662 THEN _w667 := P10D04; END_IF
D04_INT := _w667;
IF _w662 THEN _w668 := P10D05; END_IF
D05_INT := _w668;
IF _w662 THEN _w669 := P10D06; END_IF
D06_INT := _w669;
IF _w662 THEN _w670 := P10D07; END_IF
D07_INT := _w670;
IF _w662 THEN _w671 := P10D08; END_IF
D08_INT := _w671;
IF _w662 THEN _w672 := P10D09; END_IF
D09_INT := _w672;
IF _w662 THEN _w673 := P10D10; END_IF
D10_INT := _w673;
IF _w662 THEN _w674 := P10D11; END_IF
D11_INT := _w674;
IF _w662 THEN _w675 := P10D12; END_IF
D12_INT := _w675;
IF _w662 THEN _w676 := P10D13; END_IF
D13_INT := _w676;
IF _w662 THEN _w677 := P10D14; END_IF
D14_INT := _w677;
IF _w662 THEN _w678 := P10D15; END_IF
D15_INT := _w678;
IF _w662 THEN _w679 := P10D16; END_IF
D16_INT := _w679;
IF _w662 THEN _w680 := P10D17; END_IF
D17_INT := _w680;
IF _w662 THEN _w681 := P10D18; END_IF
D18_INT := _w681;
IF _w662 THEN _w682 := P10D19; END_IF
D19_INT := _w682;
IF _w662 THEN _w683 := P10D20; END_IF
D20_INT := _w683;
IF _w662 THEN _w684 := P10D21; END_IF
D21_INT := _w684;
IF _w662 THEN _w685 := P10D22; END_IF
D22_INT := _w685;
IF _w662 THEN _w686 := P10D23; END_IF
D23_INT := _w686;
IF _w662 THEN _w687 := P10D24; END_IF
D24_INT := _w687;
IF _w662 THEN _w688 := P10D25; END_IF
D25_INT := _w688;
IF _w662 THEN _w689 := P10D26; END_IF
D26_INT := _w689;
IF _w662 THEN _w690 := P10D27; END_IF
D27_INT := _w690;
IF _w662 THEN _w691 := P10D28; END_IF
D28_INT := _w691;
IF _w662 THEN _w692 := P10D29; END_IF
D29_INT := _w692;
IF _w662 THEN _w693 := P10D30; END_IF
D30_INT := _w693;
IF _w662 THEN _w694 := P10STG; END_IF
STG1_STG := _w694;

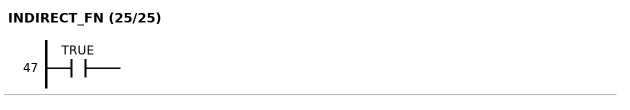
// NETWORK 47

END_FUNCTION_BLOCK

// ---- FBs/B_JKS_OldFB/Timer/fbHoldingTimer.TcPOU
FUNCTION_BLOCK fbHoldingTimer
VAR_INPUT
	bST : BOOL;
	iDelayTime : INT;
	bReset : BOOL;

END_VAR
VAR_OUTPUT
	bOutput : BOOL;
	iElapseTime : INT;

END_VAR

VAR PERSISTENT
	SecClockPls: TON;
	SecClockPlsRE: R_TRIG;
	iClockPVTime: INT;
	bOutputTime: TON;
END_VAR

SecClockPls(IN:=NOT SecClockPls.Q , PT:=t#1s , Q=> , ET=> );
SecClockPlsRE(CLK:=SecClockPls.Q , Q=> );
IF bST THEN
	IF SecClockPlsRE.Q THEN
	iClockPVTime := iClockPVTime +1;
	END_IF

	IF iDelayTime <= iClockPVTime THEN
	bOutput := TRUE;
	END_IF

END_IF

IF bReset THEN

iClockPVTime := 0;
END_IF

bOutputTime(IN:=bOutput , PT:=t#0.5s , Q=> , ET=> );

IF bOutputTime.Q THEN
iClockPVTime := 0;
bOutput := FALSE;
END_IF

iElapseTime := iDelayTime - iClockPVTime;

END_FUNCTION_BLOCK

// ---- FBs/B_JKS_OldFB/Timer/MOTION_COUNTER_RESET.TcPOU
FUNCTION_BLOCK MOTION_COUNTER_RESET
VAR_INPUT
	BOOL_JOG_ACTIVE : BOOL;
	TIME_RST_DELAY_OFF : TIME;
END_VAR
VAR_OUTPUT
	COUNTER_RST_BOOL : BOOL;
END_VAR
VAR
	DFN: F_TRIG;
	JOGDFN: BOOL;
	T1: TON;
	T1ON: BOOL;
	t0: TON;
	CUTDELAY: BOOL;
END_VAR

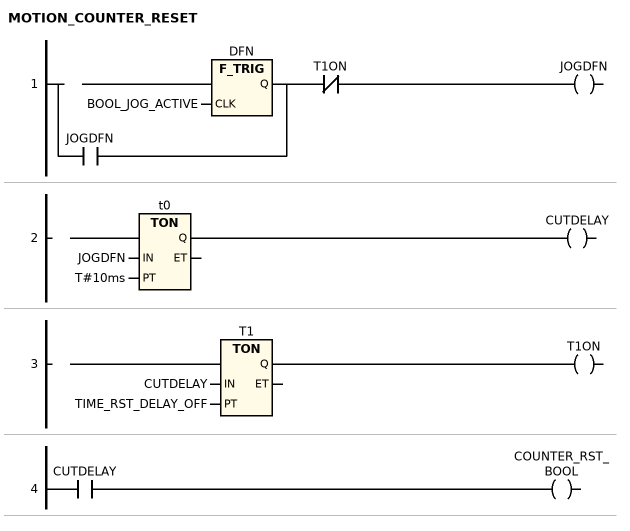
// NETWORK 1
DFN(CLK := BOOL_JOG_ACTIVE); // F_TRIG
JOGDFN := (DFN.Q OR JOGDFN) AND NOT T1ON;

// NETWORK 2
t0(IN := JOGDFN, PT := T#10ms); // TON
CUTDELAY := t0.Q;

// NETWORK 3
T1(IN := CUTDELAY, PT := TIME_RST_DELAY_OFF); // TON
T1ON := T1.Q;

// NETWORK 4
COUNTER_RST_BOOL := CUTDELAY;

END_FUNCTION_BLOCK

// ---- FBs/B_JKS_OldFB/Word to Bit/CMP_OC_DINT.TcPOU
FUNCTION_BLOCK CMP_OC_DINT
VAR_INPUT
	BOOL_INTERLOCK : BOOL; (*INTERLOCK*)
	DINT_1: DINT;		(*WORD 1*)
	END_VAR


VAR_OUTPUT
	BZ_OUTPUT_BOOL : BOOL;
END_VAR


VAR
	OUT_1: BOOL;
END_VAR

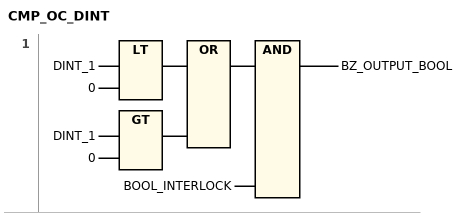
// NETWORK 1
BZ_OUTPUT_BOOL := (DINT_1 < 0 OR DINT_1 > 0) AND BOOL_INTERLOCK;

END_FUNCTION_BLOCK

// ---- FBs/B_JKS_OldFB/Word to Bit/CMP_OC_W10.TcPOU
FUNCTION_BLOCK CMP_OC_W10

VAR_INPUT
	BOOL_INTERLOCK : BOOL; (*INTERLOCK*)
	WORD_1: WORD;		(*WORD 1*)
	WORD_2: WORD;		(*WORD 2*)
	WORD_3: WORD;		(*WORD 3*)
	WORD_4: WORD;		(*WORD 4*)
	WORD_5: WORD;		(*WORD 5*)
	WORD_6: WORD;		(*WORD 6*)
	WORD_7: WORD;		(*WORD 7*)
	WORD_8: WORD;		(*WORD 8*)
	WORD_9: WORD;		(*WORD 9*)
	WORD_10: WORD;	(*WORD 10*)
END_VAR


VAR_OUTPUT
	BZ_OUTPUT_BOOL : BOOL;
END_VAR


VAR
	OUT_1: BOOL;
	OUT_2: BOOL;
	OUT_3: BOOL;
	OUT_4: BOOL;
	OUT_5: BOOL;
	OUT_6: BOOL;
	OUT_7: BOOL;
	OUT_8: BOOL;
	OUT_9: BOOL;
	OUT_10: BOOL;

END_VAR

